FUNCTION_BLOCK FB_PlantControl_mode_2
VAR_INPUT
	Start_In : BOOL;
	Stop_In : BOOL;
	Reset_In : BOOL;
END_VAR
VAR_OUTPUT
	Startet_Out : BOOL;
	Stopped_Out : BOOL;
	Reset_Out : BOOL;
END_VAR
VAR_IN_OUT
	Ctrl_Plant : Udt_PlantControl_Mode_2;
END_VAR
VAR
	SR_Start : SR;
	SR_Stop : SR;
END_VAR

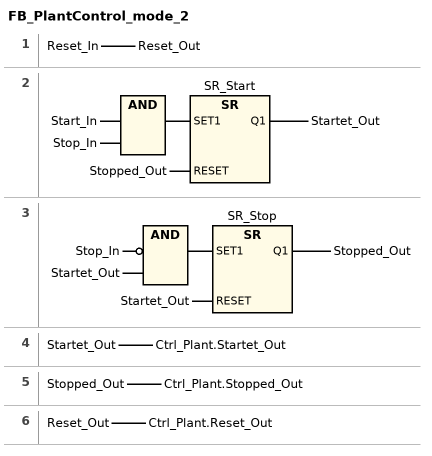
// NETWORK 1
Reset_Out := Reset_In;

// NETWORK 2
SR_Start(SET1 := Start_In AND Stop_In, RESET := Stopped_Out); // SR
Startet_Out := SR_Start.Q1;

// NETWORK 3
SR_Stop(SET1 := NOT Stop_In AND Startet_Out, RESET := Startet_Out); // SR
Stopped_Out := SR_Stop.Q1;

// NETWORK 4
Ctrl_Plant.Startet_Out := Startet_Out;

// NETWORK 5
Ctrl_Plant.Stopped_Out := Stopped_Out;

// NETWORK 6
Ctrl_Plant.Reset_Out := Reset_Out;

END_FUNCTION_BLOCK

(* stored: Version 1.1.0.1, ProductVersion 3.1.4024.13
   POU FB_PlantControl_mode_2: Id {f287aa4a-7a15-4c1e-a787-f63568e9f70c}, SpecialFunc None *)
